DATA_BLOCK "pump_flow_DB1"
{ S7_Optimized_Access := 'TRUE' }
VERSION : 0.1
NON_RETAIN
"pump_flow_set"

BEGIN

END_DATA_BLOCK

